PROGRAM Kommunikation
VAR
	Connect			:FB_ServerClientConnection;
	Connect_Local	:FB_SocketConnect;
	Listner			:FB_SocketListen;
	Accept			:FB_SocketAccept;
	Send			:FB_SocketSend;
	Receive			:FB_SocketReceive;
	LinkStatus		:FB_SocketGetLinkStatus;

	
END_VAR

VAR_INPUT
	sSrvNetID : T_AmsNetID := '';
	sLocalHost : STRING(15) := '192.168.50.10';
	nLocalPort : UDINT := 53828;
	nMode : DWORD := LISTEN_MODE_CLOSEALL (* OR CONNECT_MODE_ENABLEDBG*);
	bEnable : BOOL := TRUE;
	hServer			:T_HSERVER;
	
	eMode       : E_SocketAcceptMode := eACCEPT_SEL_HOST_PORT;
    sRemoteHost : T_IPv4Addr := '192.168.50.100';
    nRemotePort : UDINT := 30002;
    tReconnect  : TIME := T#1S;
	
	
END_VAR

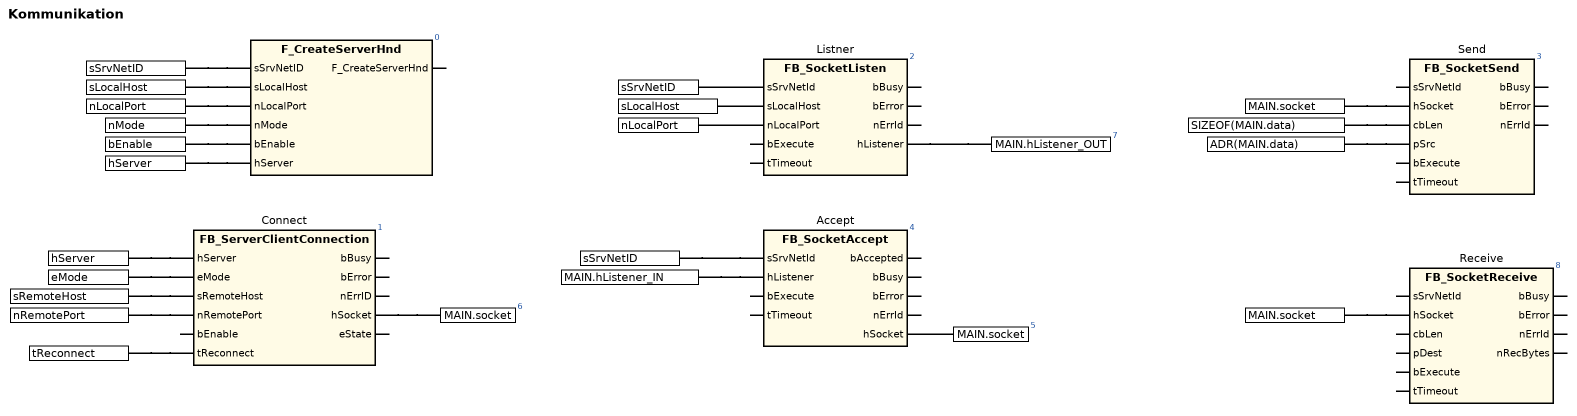
F_CreateServerHnd(sSrvNetID := sSrvNetID, sLocalHost := sLocalHost, nLocalPort := nLocalPort, nMode := nMode, bEnable := bEnable, hServer := hServer);
Connect(
    hServer := hServer,
    eMode := eMode,
    sRemoteHost := sRemoteHost,
    nRemotePort := nRemotePort,
    tReconnect := tReconnect); // FB_ServerClientConnection
Listner(sSrvNetId := sSrvNetID, sLocalHost := sLocalHost, nLocalPort := nLocalPort); // FB_SocketListen
Send(hSocket := MAIN.socket, cbLen := SIZEOF(MAIN.data), pSrc := ADR(MAIN.data)); // FB_SocketSend
Accept(sSrvNetId := sSrvNetID, hListener := MAIN.hListener_IN); // FB_SocketAccept
MAIN.socket := Accept.hSocket;
MAIN.socket := Connect.hSocket;
MAIN.hListener_OUT := Listner.hListener;
Receive(hSocket := MAIN.socket); // FB_SocketReceive

END_PROGRAM

(* stored: Version 1.1.0.1
   POU Kommunikation: Id {72a2321f-4d1d-46dc-9327-1dcc44bf5251}, SpecialFunc None *)
